//{attribute 'hide_all_locals'}
FUNCTION_BLOCK Counter EXTENDS TcoCore.TcoObject IMPLEMENTS ICounter
VAR
    _countStep  : UDINT;
    _countValue : UDINT;
    _countLimit : UDINT;

END_VAR

METHOD CountDown
_countValue := _countValue - _countStep;
END_METHOD

{attribute 'monitoring' := 'variable'}
PROPERTY CountLimitReached : BOOL
GET
CountLimitReached := CountValue >= _countLimit;
END_GET
END_PROPERTY

METHOD CountUp

_countValue := _countValue + _countStep;
END_METHOD

{attribute 'monitoring' := 'monitor'}
PROPERTY CountValue : UDINT
GET
CountValue := _countValue;
END_GET
END_PROPERTY

{attribute 'monitoring' := 'variable'}
PROPERTY CountZeroReached : BOOL
GET
CountZeroReached:= CountValue = 0;
END_GET
END_PROPERTY

{attribute 'hide'}
METHOD FB_init : BOOL
VAR_INPUT
    (* if TRUE, the retain variables are initialized (warm start / cold start)*)
    bInitRetains : BOOL;
    (* if TRUE, the instance afterwards gets moved into the copy code (online change)*)
    bInCopyCode  : BOOL;
    ParentObject : ITcoObject;

    countStep      : UDINT;
    countInitValue : UDINT;
    countLimit     : UDINT;
END_VAR
//SUPER^.FB_init(bInitRetains, bInCopyCode, ParentObject);

_countStep := countStep;
_countValue := countInitValue;
_countLimit := countLimit;

IF countInitValue > countLimit THEN
    Messenger.Error('Value groesser als Limit eingestellt');
    RETURN;
END_IF
END_METHOD

METHOD ResetCount
_countValue := 0;
END_METHOD

END_FUNCTION_BLOCK

(* stored: Version 1.1.0.1, ProductVersion 3.1.4024.12
   POU Counter: Id {71761be2-846a-03d7-24fd-9df14ef6de76}, SpecialFunc None
   Method CountDown: Id {fbcebd65-b073-042c-0580-9caf1d87a402}
   Property CountLimitReached: Id {6ff381d1-d150-0405-3307-973197abea7c}
   Get Get: Id {11a815fc-0412-04bf-3c78-7cb2d56e0265}
   Method CountUp: Id {0689e83a-e86c-036c-1fad-26a429474485}
   Property CountValue: Id {a47fbf65-5553-03b4-133f-2092def58893}
   Get Get: Id {dbf8f875-581e-013c-00bf-04ea6089a5c1}
   Property CountZeroReached: Id {14fe20d1-0de4-01e8-1131-c439570199b8}
   Get Get: Id {45620290-2679-0cc7-0d31-412975b1e6e6}
   Method FB_init: Id {d430239b-e232-0b79-2b53-93e5164e2e76}
   Method ResetCount: Id {6ec835ed-0aaa-0362-2dbc-f1eaa28343ce} *)
